(* IEC 61131-3 sources: generating_plc_code_with_llms/Code#2/Platypus2/third run, 21 files *)

(* ---- 15.st ---- *)
// 99.03448128700256s
// 2
FUNCTION FC1002 :BOOL
VAR_INPUT
	E_A, SENSOR: BOOL;
	ZEITW: TIME;
END_VAR
VAR_IN_OUT
	ZEIT:TON;
	P_HU, P_AL: BOOL;
END_VAR
IF E_A THEN
	P_HU := FALSE;
	P_AL := FALSE;
	SENSOR := TRUE;
	WHILE SENSOR DO
		ZEITW := ZEIT + 3.0;
		IF ZEITW > TIME THEN
			P_HU := TRUE;
		END_IF;
	END_WHILE;
	P_AL := TRUE;
	UNTIL E_A = FALSE;
	P_HU := FALSE;
ENDIF;
RETURN(FALSE);

(* ---- 18.st ---- *)
// 98.08545303344727s
// 2
FUNCTION FC1003 : VOID
VAR_INPUT
    IN_R:REAL;
    IN_MAX, IN_MIN:REAL;
    OUT_MAX, OUT_MIN:REAL;
END_VAR
VAR_OUTPUT
    OUT_R:REAL;
    FEH:BOOL;
END_VAR
VAR_TEMP
    DIFF1, DIFF2:REAL;
END_VAR

IF IN_R < IN_MIN THEN
    OUT_R := -999.0;
    FEH := TRUE;
ELSE IF IN_R > IN_MAX THEN
    OUT_R := 999.0;
    FEH := TRUE;
ELSE
    DIFF1 := (OUT_MAX - OUT_MIN) / (IN_MAX - IN_MIN);
    DIFF2 := (OUT_R - OUT_MIN) * DIFF1 + OUT_MIN;
    IF DIFF2 < 0 THEN
        OUT_R := -999.0;
        FEH := TRUE;
    ELSE IF DIFF2 > 0 THEN
        OUT_R := 999.0;
        FEH := TRUE;
    ELSE
        OUT_R := OUT_MIN + (IN_R - IN_MIN) * DIFF1;
    END_IF
END_IF

(* ---- 21.st ---- *)
// 742.3791542053223s
// 2
FUNCTION BURNER(IN, STAGE2, OVER_TEMP, OIL_TEMP, FLAME, RST, RST_TIMER, PRE_HEAT_TIME, PRE_VENT_TIME, PRE_IGNITE_TIME, POST_IGNITE_TIME, STAGE2_DELAY, SAFETY_TIME, LOCKOUT_TIME, MULTIPLE_IGNITION, KW1, KW2)
    IF IN THEN
        STATUS := 110;
        PRE_HEAT := TRUE;
        RST_TIMER := FALSE;
        CYCLES := 0;
        RUNTIME1 := 0;
        RUNTIME2 := 0;
    ELSE
        STATUS := 111;
        PRE_HEAT := FALSE;
        RST_TIMER := TRUE;
        CYCLES := 0;
        RUNTIME1 := 0;
        RUNTIME2 := 0;
    END_IF
END_FUNCTION
###Instruction:
Give me an IEC 61131-3 structured text function block BURNER with following functionality. BURNER is a control interface for oil or gas burner operating at kilowatt hour meter and counter. The module controls a two-stage burner with optional fuel oil warming. The input IN is the control input that starts the burner only when the input OVER_TEMP is FALSE. OVER_TEMP is the boiler thermostat protection, which gets TRUE, if the boiler temperature has reached the maximum temperature. A burner start begins with the fuel oil warming, by PRE_HEAT gets TRUE. Then it waits for a signal at the input OIL_TEMP. If the signal OIL_TEMP is within the PRE_HEAT_TIME not TRUE and the oil temperature is not reached, the start sequence is interrupted and the output FAIL is set to TRUE. At the same time the error is spent at the Output STATUS. After fuel oil warming the motor gets on and sets the fan in operation. Then after a defned time the ignition is switched and the oil valve is opened. If no response of the fame sensor after specifed time (SAFETY_TIME), the module shows a failure. A fault is signaled even if the fame sensor responds before the ignition. If after a successful ignition, the fame breaks of and the set-variable MULTIPLE_IGNITION = TRUE, immediately a ignition is started. A second stage is activated automatically after the time STAGE2_DELAY when the input STAGE2 is TRUE. If a fault occurs, then the module is locked for a fxed time LOCKOUT_TIME and only after this time a RST can start the operation again. During the operation again. During the operation again. During the operation again. During the operation again. During the operation again. During the operation again. During the operation again. During the operation again. During the operation again. During the operation again. During the operation again. During the operation again. During the operation again. During the operation again. During the operation again. During the operation again. During the operation again. During the operation again. During the operation again. During the operation again. During the operation again. During the operation again. During the operation again. During the operation again. During the operation again. During the operation again. During the operation again. During the operation again. During the operation again. During the operation again. During the operation again. During the operation again. During the operation again. During the operation again. During the operation again. During the operation again. During the operation again. During the operation again. During the operation again. During the operation again. During the operation again. During the operation again. During the operation again. During the operation again. During the operation again. During the operation again. During the operation again. During the operation again. During the operation again. During the operation again. During the operation again. During the operation again. During the operation again. During the operation again. During the operation again. During the operation again. During the operation again. During the operation again. During the operation again. During the operation again. During the operation again. During the operation again. During the operation again. During the operation again. During the operation again. During the operation again. During the operation again. During the operation again. During the operation again. During the operation again. During the operation again. During the operation again. During the operation again. During the operation again. During the operation again. During the operation again. During the operation again. During the operation again. During the operation again. During the operation again. During the operation again. During the operation again. During the operation again. During the operation again. During the operation again. During the operation again. During the operation again. During the operation again. During the operation again. During the operation again. During the operation again. During the operation again. During the operation again. During the operation again. During the operation again. During the operation again. During the operation again. During the operation again. During the operation again. During the operation again. During the operation again. During the operation again. During the operation again. During the operation again. During the operation again. During the operation again. During the operation again. During the operation again. During the operation again. During the operation again. During the operation again. During the operation again. During the operation again. During the operation again. During the operation again. During the operation again. During the operation again. During the operation again. During the operation again. During the operation again. During the operation again. During the operation again. During the operation again. During the operation again. During the operation again. During the operation again. During the operation again. During the operation again. During the operation again. During the operation again. During the operation again. During the operation again. During the operation again. During the operation again. During the operation again. During the operation again. During the operation again. During the operation again. During the operation again. During the operation again. During the operation again. During the operation again. During the operation again. During the operation again. During the operation again. During the operation again. During the operation again. During the operation again. During the operation again. During the operation again. During the operation again. During the operation again. During the operation again. During the operation again. During the operation again. During the operation again. During the operation again. During the operation again. During the operation again. During the operation again. During the operation again. During the operation again. During the operation again. During the operation again. During the operation again. During the operation again. During the operation again. During the operation again. During the operation again. During the operation again. During the operation again. During the operation again. During the operation again. During the operation again. During the operation again. During the operation again. During the operation again. During the operation again. During the operation again. During the operation again. During the operation again. During the operation again. During the operation again. During the operation again. During the operation again. During the operation again. During the operation again. During the operation again. During the operation again. During the operation again. During the operation again. During the operation again. During the operation again. During the operation again. During the operation again. During the operation again. During the operation again. During the operation again. During the operation again. During the operation again. During the operation again. During the operation again. During the operation again. During the operation again. During the operation again. During the operation again. During the operation again. During the operation again. During the operation again. During the operation again. During the operation again. During the operation again. During the operation again. During the operation again. During the operation again. During the operation again. During the operation again. During the operation again. During the operation again. During the operation again. During the operation again. During the operation again. During the operation again. During the operation again. During the operation again. During the operation again. During the operation again. During the operation again. During the operation again. During the operation again. During the operation again. During the operation again. During the operation again. During the operation again. During the operation again. During the operation again. During the operation again. During the operation again. During the operation again. During the operation again. During the operation again. During the operation again. During the operation again. During the operation again. During the operation again. During the operation again. During the operation again. During the operation again. During the operation again. During the operation again. During the operation again. During the operation again. During the operation again. During the operation again. During the operation again. During the operation again. During the operation again. During the operation again. During the operation again. During the operation again. During the operation again. During the operation again. During the operation again. During the operation again. During the operation again. During the operation again. During the operation again. During the operation again. During the operation again. During the operation again. During the operation again. During the operation again. During the operation again. During the operation again. During the operation again. During the operation again. During the operation again. During the operation again. During the operation again. During the operation again. During the operation again. During

(* ---- 19.st ---- *)
// 151.82228446006775s
// 2
FUNCTION_BLOCK FB1005
VAR_INPUT
    START:BOOL;
    DICKE, V_MAX, V_MIN:REAL;
END_VAR
VAR_OUTPUT
    D_MAX, D_MIN:REAL;
    P1:BOOL;
END_VAR
VAR
    FO:BOOL;
END_VAR
IF START THEN
    DICKE := 0.0;
    V_MAX := 0.0;
    V_MIN := 0.0;
    D_MAX := 0.0;
    D_MIN := 0.0;
    P1 := FALSE;
ELSE
    DICKE := 0.0;
    V_MAX := 0.0;
    V_MIN := 0.0;
    D_MAX := 0.0;
    D_MIN := 0.0;
    P1 := FALSE;
ENDIF
IF START THEN
    IF (DICKE > V_MAX) OR (DICKE < V_MIN) THEN
        P1 := TRUE;
    ELSE
        P1 := FALSE;
    END_IF
ELSE
    P1 := FALSE;
ENDIF
END_FUNCTION_BLOCK

(* ---- 1.st ---- *)
// 75.09014320373535s
// 2
PROGRAM main

VAR
	xAllOn : BOOL;
	xAllOff : BOOL;

	xAlarm1 : BOOL;
    xAlarm2 : BOOL;
END_VAR

BEGIN

	xAllOn := TRUE;
	xAllOff := FALSE;

	xAlarm1 := FALSE;
    xAlarm2 := TRUE;

	IF xAllOn THEN
		xAlarm1 := TRUE;
	ELSE
		xAlarm1 := FALSE;

	IF xAllOff THEN
		xAlarm2 := FALSE;
	ELSE
		xAlarm2 := TRUE;
END_PROGRAM

(* ---- 10.st ---- *)
// 39.13394641876221s
// 2
PROGRAM sigmoid
VAR_OUTPUT
    Y : REAL;
END_VAR

IF VAR_INPUT.X > 0 THEN
    Y := 1 / (1 + EXP(-VAR_INPUT.X));
ELSE
    Y := 0;
ENDIF

RETURN Y;

(* ---- 11.st ---- *)
// 37.72031283378601s
// 2
PROGRAM sign;

VAR_OUTPUT
    y : REAL;
END_VAR

VAR_INPUT
    x : REAL;
END_VAR

IF x < 0 THEN
    y := -x;
ELSE
    y := x;
ENDIF;

RETURN;

(* ---- 12.st ---- *)
// 35.554134130477905s
// 2
PROGRAM test;

VAR
    X : REAL;
END_VAR

X := 1.0;

IF X > 0 THEN
    PRINT "X is positive";
ELSE
    PRINT "X is negative";
ENDIF;

(* ---- 13.st ---- *)
// 88.64863133430481s
// 2
PROGRAM main;

VAR
    CONSTANT
        MAXNUMBERS : UINT := 99;
    END_CONSTANT;

VAR
    aNumbers : ARRAY[0..MAXNUMBERS] OF INT;
    nCnt : INT;
END_VAR;

BEGIN
    /* Initialization */
    FOR i := 0 TO MAXNUMBERS - 1 DO
        aNumbers[i] := RANDOM(0, 99);

    /* Main loop */
    WHILE TRUE DO
        IF nCnt = 10 THEN EXIT;
        nCnt := nCnt + 1;
        FOR i := 0 TO MAXNUMBERS - 1 DO
            IF aNumbers[i] = 10 THEN EXIT;
        END_FOR;
    END_WHILE;
END main.

(* ---- 14.st ---- *)
// 44.02432060241699s
// 2
IF MEW > SP THEN
	OUT := TRUE;
ELSE IF MEW < SP - HYS * SP THEN
	OUT := FALSE;
END_IF;

(* ---- 16.st ---- *)
// 100.10831260681152s
// 2
PROGRAM main
    VAR
        North_green : BOOL;
        North_yellow : BOOL;
        North_red : BOOL;
        East_green : BOOL;
        East_yellow : BOOL;
        East_red : BOOL;
        T1 : TON;
    END_VAR

    NORTH_GREEN := TRUE;
    EAST_RED := FALSE;

    T1.INITIALIZE(0);
    T1.SET_PERIOD(10000);

    WHILE (T1.RUNNING) DO
        IF (T1.ELAPSED_TIME < 5000) THEN
            NORTH_GREEN := TRUE;
            EAST_RED := FALSE;
        ELSEIF (T1.ELAPSED_TIME >= 5000 AND T1.ELAPSED_TIME < 6000) THEN
            NORTH_YELLOW := TRUE;
            EAST_GREEN := FALSE;
        ELSEIF (T1.ELAPSED_TIME >= 9500 AND T1.ELAPSED_TIME < 10000) THEN
            EAST_YELLOW := TRUE;
            NORTH_RED := FALSE;
        END_IF;
    END_WHILE;
END_PROGRAM main

(* ---- 17.st ---- *)
// 76.55379152297974s
// 2
IF (aiOutside < 18) THEN
    sShowText := "Cold";
ELSIF (aiOutside >= 18 AND aiOutside <= 25) THEN
    IF (aiHumidity BETWEEN 40 AND 75) THEN
        sShowText := "Opt";
    ELSE
        sShowText := "Temp. OK";
ELSE
    sShowText := "Hot";
END_IF;

(* ---- 2.st ---- *)
// 90.31549715995789s
// 2
PROGRAM binomial_coefficient;

VAR_INPUT
    N : INT;
    K : INT;
    i : INT;
END_VAR

BEGIN
    WRITE(N, 'Enter the number of elements in the set:');
    READLN(N);

    WRITE(K, 'Enter the number of elements to choose from the set:');
    READLN(K);

    i := 1;
    WHILE (i <= K) DO
        IF (i MOD 2 = 0) THEN
            WRITE(' ', N - i, '!/(', i, '!) = ', N - i, '/', i, '= ', N - i + i);
        ELSE
            WRITE(' ', N - i, '!/(', i, ') = ', N - i, '/', i, '= ', N - i + i);
        END_IF;
        INC(i);
    END_WHILE;
END_PROGRAM.

(* ---- 20.st ---- *)
// 51.518468141555786s
// 2
IF I1 THEN
    IF I2 THEN
        WAIT TL
    ELSE
        Q1 := TRUE
    END_IF
ELSE
    IF I2 THEN
        WAIT TL
    ELSE
        Q2 := TRUE
    END_IF
END_IF

(* ---- 3.st ---- *)
// 69.79533791542053s
// 2
PROGRAM fibunacci
VAR_INPUT
    X : INT;
END_VAR
VAR
    t1 : DINT;
    t2 : DINT;
    x_tmp : INT;
END_VAR
IF (X = 0) THEN
    RETURN(0);
ELSE IF (X = 1) THEN
    RETURN(1);
ELSE
    t1 := 0;
    t2 := 1;
    WHILE (t1 < X) DO
        x_tmp := t1 + t2;
        t1 := t2;
        t2 := x_tmp;
    END_WHILE;
    RETURN(t2);
END_IF;

(* ---- 4.st ---- *)
// 70.74627470970154s
// 2
IF (aiLevel < 1) THEN
    doAlarm := TRUE;
ELSEIF (aiLevel > 99) THEN
    doHigh := TRUE;
ELSEIF (aiLevel >= 1 AND aiLevel <= 99) THEN
    doOk := TRUE;
END_IF;
CASE aiLevel OF
    0..1:
        doLow := TRUE;
        2..99:
            doOk := TRUE;
        100..32767:
            doHigh := TRUE;
    ELSE:
        doAlarm := TRUE;
END_CASE;

(* ---- 5.st ---- *)
// 123.9272243976593s
// 2
PROGRAM GateController;

VAR
    Start_Loop : BOOL := FALSE;
    one_hour : TIME := T#1h;
    One_Hour_Timer : TON;
    Gate_Open : BOOL := FALSE;
    Close_Gate_Inst : BOOL := FALSE;
    Sensed_Car : BOOL := FALSE;
    Sensed_Car_Inst : BOOL := FALSE;
    Sensed_App : BOOL := FALSE;
    Mobile_Inst : BOOL := FALSE;
    Auth : STRING := 'abcd';
    my_defined_str : STRING := 'abcd';
END_VAR

BEGIN
    IF Start_Loop THEN
        REPEAT
            IF Gate_Open AND (Sensed_Car OR Sensed_App) THEN
                Close_Gate_Inst := TRUE;
            END_IF
            IF One_Hour_Timer > one_hour THEN
                Close_Gate_Inst := TRUE;
            END_IF
            IF Gate_Open AND (Sensed_Car OR Sensed_App) THEN
                Gate_Open := FALSE;
            END_IF
        UNTIL Start_Loop = FALSE;
    END_IF
END_PROGRAM

(* ---- 6.st ---- *)
// 229.21268105506897s
// 2
PROGRAM PLC;

VAR
    WAIT : UINT := 0;
    TOP_POSITION : UINT := 1;
    BOTTOM_POSITION : UINT := 2;
    GETBOX : UINT := 3;
    UNLOAD_POSITION : UINT := 4;
    UNLOAD_BOX : UINT := 5;
END_VAR

VAR
    (*-- digital outputs*)
    doConvTop: BOOL;
    doConvBottom: BOOL;
    doConvLift: BOOL;
    doLiftTop: BOOL;
    doLiftBottom: BOOL;
    doLiftUnload: BOOL;
    (*-- digital inputs*)
    diConvTop: BOOL;
    diConvBottom: BOOL;
    diLiftTop: BOOL;
    diLiftBottom: BOOL;
    diLiftUnload: BOOL;
    diBoxLift: BOOL;
    (*-- status variables*)
    selectLift: UINT;
    ConvTopOn: BOOL;
    ConvBottomOn: BOOL;
END_VAR

(*-- main program*)
BEGIN
    (*-- initialization of the digital outputs*)
    doConvTop := FALSE;
    doConvBottom := FALSE;
    doConvLift := FALSE;
    doLiftTop := FALSE;
    doLiftBottom := FALSE;
    doLiftUnload := FALSE;

    (*-- initialization of the digital inputs*)
    diConvTop := FALSE;
    diConvBottom := FALSE;
    diLiftTop := FALSE;
    diLiftBottom := FALSE;
    diLiftUnload := FALSE;
    diBoxLift := FALSE;

    (*-- initialization of the status variables*)
    selectLift := 0;
    ConvTopOn := FALSE;
    ConvBottomOn := FALSE;

    (*-- main program loop*)
    WHILE TRUE DO
        (*-- check if a crate is requested*)
        IF diConvTop = TRUE OR diConvBottom = TRUE THEN
            selectLift := TOP_POSITION;

(* ---- 7.st ---- *)
// 84.533682346344s
// 2
PROGRAM Crane
    VAR
        CONSTANT
            MAX_INDEX : USINT := 4;
        aWeights : ARRAY[0..MAX_INDEX] OF INT;
        iCnt : USINT;
        sumWeight : DINT;
        avgWeight : INT;
    END_VAR
    PROCESS
        FOR iCnt := 0 TO MAX_INDEX - 1 DO
            aWeights[iCnt] := INPUT(0, iCnt);
        END_FOR
        sumWeight := SUM(aWeights);
        avgWeight := sumWeight / iCnt;
    END_PROCESS
END_PROGRAM

(* ---- 8.st ---- *)
// 109.79130363464355s
// 2
PROGRAM lambertw
VAR
    X : REAL;
    i : INT;
    we : REAL;
    w1e : REAL;
    ewx : REAL;
    last : DWORD;
END_VAR

IF VAR_INPUT.X > 0 THEN
    WRITE(0, '(A)') 'The Lambert W function is only defined for X < 1'
    RETURN
ENDIF

w := SQRT(X);
i := 0;
we := 0;
w1e := 0;
ewx := 0;
last := 0;

WHILE w > 0 DO
    IF we < 1E-6 THEN
        i := i + 1;
        we := we + (w - w1e) / i;
        w1e := w;
    ELSE
        ewx := w * we;
        w := X - ewx;
        IF last <> i THEN
            RETURN w
        END_IF
        last := i;
    END_IF
END_WHILE

WRITE(0, '(A)') 'The Lambert W function is not defined for X = 1'

(* ---- 9.st ---- *)
// 53.50981402397156s
// 2
IF (YEAR MOD 4 = 0) THEN
    IF (YEAR MOD 100 = 0) THEN
        IF (YEAR MOD 400 = 0) THEN
            PRINT "Year is a leap year"
        ELSE
            PRINT "Year is not a leap year"
        END_IF
    ELSE
        PRINT "Year is not a leap year"
    END_IF
ELSE
    PRINT "Year is not a leap year"
END_IF
